TYPE ST_OuputStationHSAdditionalDataOP11600 :
STRUCT
	{attribute 'OPC.UA.DA.Description' := 'Dummy (for making struct visible on OPC UA'}
	Dummy						: BOOL;
END_STRUCT
END_TYPE

(* stored: Version 1.1.0.1, ProductVersion 3.1.4024.2
   DUT ST_OuputStationHSAdditionalDataOP11600: Id {d89dff96-7d05-4b65-9fe4-92a420618f67} *)
